// TIA Portal V19 export
FUNCTION_BLOCK "TYPIC_C403_IF_SOS"   // FB118, FBD
TITLE = TYPIC_C403_IF_SOS: Snelheidsonderschrijding
{ S7_Optimized_Access := 'TRUE' }
AUTHOR : OCOTECH
FAMILY : Typical
NAME : C403.701
// Logisch Object Besturing: C403.701
// 
// Het doel van de IF SOS (SnelheidsOnderschrijdingsSysteem) is om de algemene gegevens te verwerken die ontvangen worden vanuit de interne sturing en via inputs.
// stored: MemoryReserve 10, SetENOAutomatically false
   VAR_INPUT
      EXT_HW { ExternalAccessible := 'False'; ExternalVisible := 'False'; ExternalWritable := 'False'} : Bool;   // Sturings hardware (PLC) bewaking (1 = OK)
      IN_AUT_C403 { ExternalAccessible := 'False'; ExternalVisible := 'False'; ExternalWritable := 'False'} : Bool;   // Beveiligingen: serie geschakelde terugmelding (1= OK)
      IN_STO { ExternalAccessible := 'False'; ExternalVisible := 'False'; ExternalWritable := 'False'} : Word;   // Algemene storingen
   END_VAR
   VAR_OUTPUT
      VAR_IF_SOS { ExternalAccessible := 'False'; ExternalVisible := 'False'; ExternalWritable := 'False'} : "C403_VAR_IF_SOS_TYPIC";   // Struct met alle variabelen naar de basisfunctie
   END_VAR
   VAR
      STO { ExternalWritable := 'False'} : Struct   // Storingen
         A001 : Bool;   // Beveiliging aangesproken
         A002 : Bool;   // SOS-detectie is over 60 m tot 150 m uitgevallen
         A003 : Bool;   // SOS-detectie is over meer dan 150 m uitgevallen
      END_STRUCT;
      VAR { ExternalWritable := 'False'} : Struct   // Variabelen
         EXT_HW { ExternalAccessible := 'False'; ExternalVisible := 'False'} : Bool;   // Sturings hardware (PLC) in storing
      END_STRUCT;
   END_VAR
BEGIN

REGION Network 1: START
END_REGION

REGION Network 2: +++ Storingen +++
   // Verzamelen storingsmeldingen.
END_REGION

REGION Network 3: Storing A001: Beveiliging aangesproken
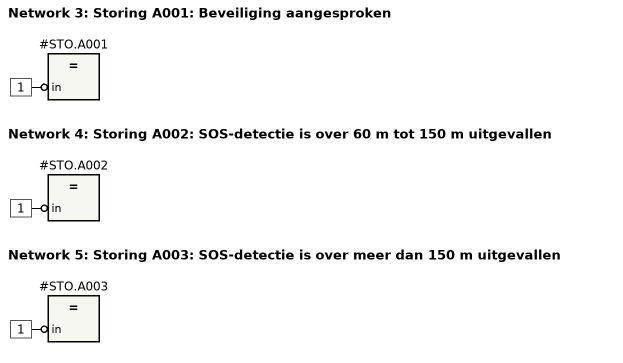
   #STO.A001 := NOT 1;
END_REGION

REGION Network 4: Storing A002: SOS-detectie is over 60 m tot 150 m uitgevallen
   #STO.A002 := NOT 1;
END_REGION

REGION Network 5: Storing A003: SOS-detectie is over meer dan 150 m uitgevallen
   #STO.A003 := NOT 1;
END_REGION

REGION Network 6 (SCL): EINDE
   // Variabelen van intern scada rakvlak naar outputs copieren
   #VAR_IF_SOS.EXT_HW := #VAR.EXT_HW;
   #VAR_IF_SOS.STO := #STO;
END_REGION
END_FUNCTION_BLOCK
